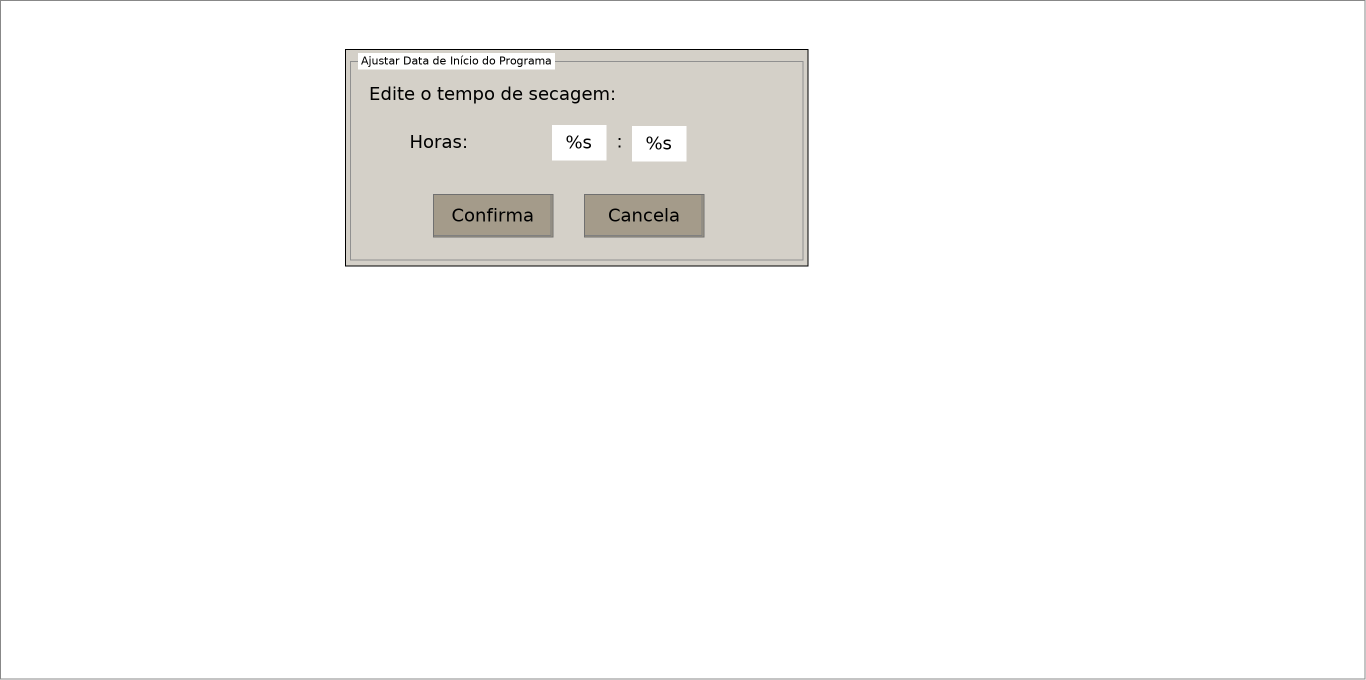
VISUALIZATION setSecagem  // 1366x680
    Rectangle (345,49 463x217)
    GroupBox (350,53 453x207), "Ajustar Data de Início do Programa"
        Label (16,25 316x32), "Edite o tempo de secagem:"
        Textfield (201,71 56x37), "%s", text variable: GVL.horaSecagem
            OnMouseClick: write the text variable via VisuDialogs.Numpad
        Textfield (281,72 56x37), "%s", text variable: GVL.minSecagem
            OnMouseClick: write the text variable via VisuDialogs.Numpad
        Label (35,74 86x30), "Horas:"
        Label (258,71 23x35), ":"
        Button (83,141 120x43), "Confirma"
            OnMouseClick: CloseDialog Dialog=setSecagem, Result=OK, NumpadKeypadSet=True
            OnMouseClick: execute { confirmSetInicio(); }
        Button (234,141 120x43), "Cancela"
            OnMouseClick: CloseDialog Dialog=setSecagem, Result=Cancel, NumpadKeypadSet=True
END_VISUALIZATION

(* stored: Version 1.1.0.1, ProductVersion 3.1.4024.12
   Visu setSecagem: Id {0cfe1076-8a99-409c-ad58-14977d37a597} *)
